TYPE GearOut_Statuses_typ EXTENDS MultiAxis_Status_typ:
	STRUCT
		

	END_STRUCT
END_TYPE

(* stored: Version 1.1.0.1, ProductVersion 3.1.4024.3
   DUT GearOut_Statuses_typ: Id {c55deee6-6cc9-0643-3574-88c1109fb23f} *)
